// TIA Portal V17 export
// export: Created 2022-06-21T13:51:02.5238312Z, ExportSetting WithDefaults, DisplayName Totally Integrated Automation Portal, DisplayVersion V17, DisplayName TIA Portal Openness, DisplayVersion V17, DisplayName TIA Portal Version Control Interface, DisplayVersion V17, DisplayName STEP 7 Professional, DisplayVersion V17, DisplayName STEP 7 Safety, DisplayVersion V17, DisplayName WinCC Advanced, DisplayVersion V17
VAR_GLOBAL   // PLC tag table "MotionControl_Tag table"
END_VAR
VAR_GLOBAL CONSTANT   // user constants
   AXIS_NUM : Int := 3;
   TEST_VECTOR_NUM : Int := 10;
END_VAR
